TYPE ST_HmiControl :
STRUCT
	fTargetPosition : LREAL;
	fVelocity : LREAL := 100;
	fFwdLimit : LREAL;
	fBwdLimit : LREAL;
	fLocalModeSpeedOverride : LREAL;
END_STRUCT
END_TYPE

(* stored: Version 1.1.0.1, ProductVersion 3.1.4024.11
   DUT ST_HmiControl: Id {af3cd7ba-0cc2-4c79-b8f0-e738ae733380} *)
